// Mitsubishi GX Works2 project: 增加消防20180613   PLC: FX3G

PROGRAM MAIN
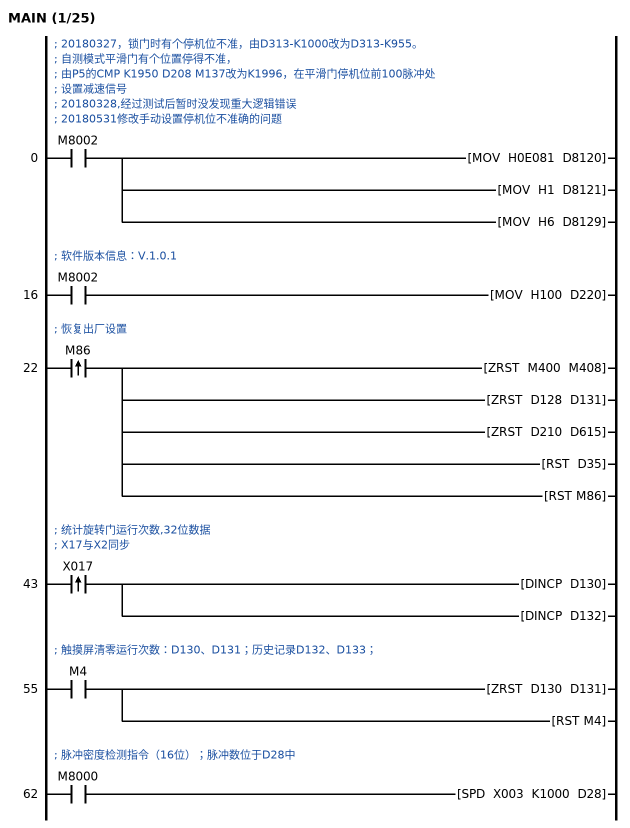
; 20180327，锁门时有个停机位不准，由D313-K1000改为D313-K955。
; 自测模式平滑门有个位置停得不准，
; 由P5的CMP K1950 D208 M137改为K1996，在平滑门停机位前100脉冲处
; 设置减速信号
; 20180328,经过测试后暂时没发现重大逻辑错误
; 20180531修改手动设置停机位不准确的问题
0     LD      M8002
      MOV     H0E081 D8120
        [note] 设置通讯方式
      MOV     H1 D8121
        [note] 站号设置：01H
      MOV     H6 D8129
        [note] 超时检查时间60ms
; 软件版本信息：V.1.0.1
16    LD      M8002
      MOV     H100 D220
        [note] V.1.0.1
; 恢复出厂设置
22    LDP     M86
      ZRST    M400 M408
      ZRST    D128 D131
      ZRST    D210 D615
      RST     D35
      RST     M86
; 统计旋转门运行次数,32位数据
; X17与X2同步
43    LDP     X017
      DINCP   D130
      DINCP   D132
; 触摸屏清零运行次数：D130、D131；历史记录D132、D133；
55    LD      M4
      ZRST    D130 D131
      RST     M4
; 脉冲密度检测指令（16位）；脉冲数位于D28中
62    LD      M8000
      SPD     X003 K1000 D28
        [note] 速度检测
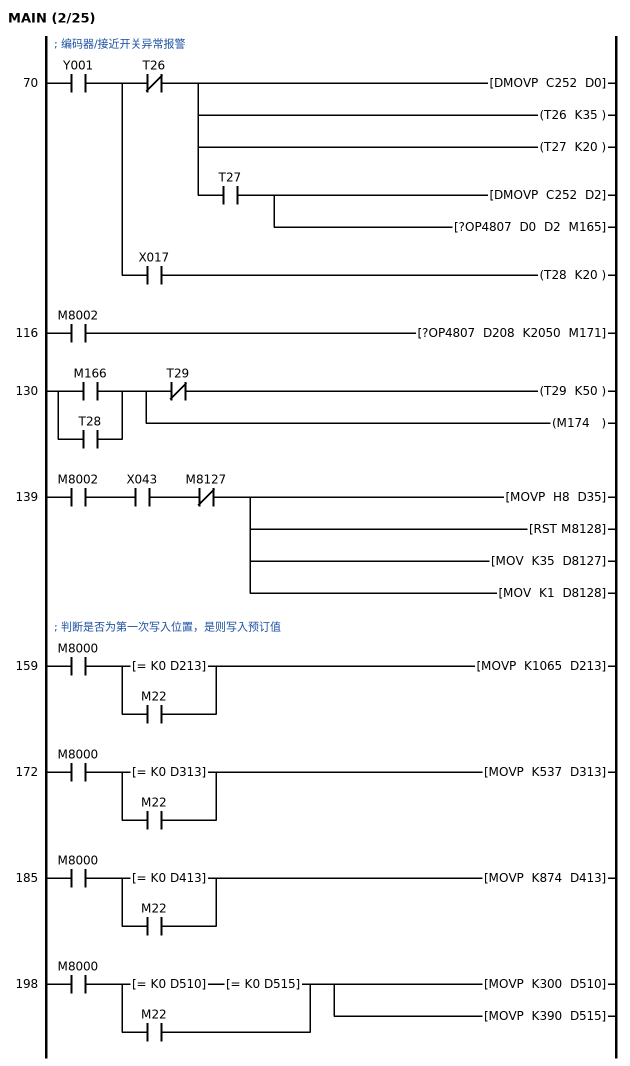
; 编码器/接近开关异常报警
70    LD      Y001
      MPS
      ANI     T26
      DMOVP   C252 D0
      OUT     T26 K35
      OUT     T27 K20
      AND     T27
      DMOVP   C252 D2
      ?OP4807 D0 D2 M165
        [note] Y1=1时，D0D1=D2D3，编码器坏
      MPP
      AND     X017
      OUT     T28 K20
        [note] Y1=1时，编码器连续2s清零0，坏
116   LD      M8002
      ?OP4807 D208 K2050 M171
        [note] 编码器值>2050时M173置位
130   LD      M166
      OR      T28
      MPS
      ANI     T29
      OUT     T29 K50
        [note] 每隔5秒发送一次报警命令
      MPP
      OUT     M174
139   LD      M8002
      AND     X043
      ANI     M8127
      MOVP    H8 D35
      RST     M8128
      MOV     K35 D8127
      MOV     K1 D8128
; 判断是否为第一次写入位置，是则写入预订值
159   LD      M8000
      LD=     K0 D213
      OR      M22
      ANB
      MOVP    K1065 D213
        [note] 平滑门位置
172   LD      M8000
      LD=     K0 D313
      OR      M22
      ANB
      MOVP    K537 D313
        [note] 冬季位置
185   LD      M8000
      LD=     K0 D413
      OR      M22
      ANB
      MOVP    K874 D413
        [note] 夏季位置
198   LD      M8000
      LD=     K0 D510
      AND=    K0 D515
      OR      M22
      ANB
      MOVP    K300 D510
        [note] 危险区域1
      MOVP    K390 D515
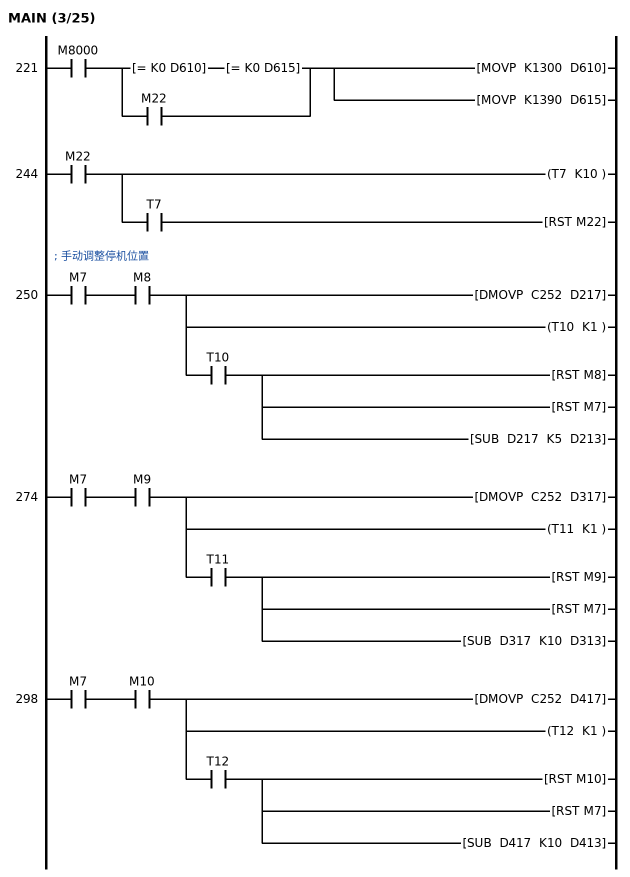
221   LD      M8000
      LD=     K0 D610
      AND=    K0 D615
      OR      M22
      ANB
      MOVP    K1300 D610
        [note] 危险区域2
      MOVP    K1390 D615
244   LD      M22
      OUT     T7 K10
      AND     T7
      RST     M22
; 手动调整停机位置
250   LD      M7
      AND     M8
      DMOVP   C252 D217
        [note] 手动调整平滑模式参考位
      OUT     T10 K1
      AND     T10
      RST     M8
      RST     M7
      SUB     D217 K5 D213
274   LD      M7
      AND     M9
      DMOVP   C252 D317
        [note] 手动调整冬季模式参考位
      OUT     T11 K1
      AND     T11
      RST     M9
      RST     M7
      SUB     D317 K10 D313
298   LD      M7
      AND     M10
      DMOVP   C252 D417
        [note] 手动调整夏季模式参考位
      OUT     T12 K1
      AND     T12
      RST     M10
      RST     M7
      SUB     D417 K10 D413
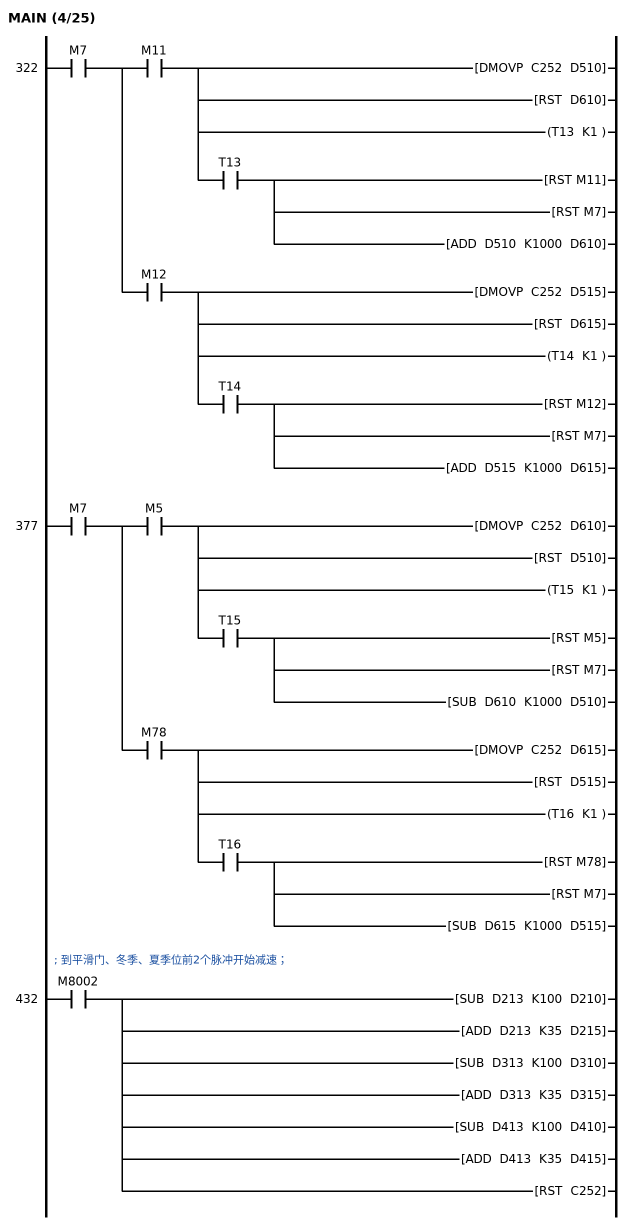
322   LD      M7
      MPS
      AND     M11
      DMOVP   C252 D510
        [note] 手动调危险区1参考位
      RST     D610
      OUT     T13 K1
      AND     T13
      RST     M11
      RST     M7
      ADD     D510 K1000 D610
      MPP
      AND     M12
      DMOVP   C252 D515
      RST     D615
      OUT     T14 K1
      AND     T14
      RST     M12
      RST     M7
      ADD     D515 K1000 D615
377   LD      M7
      MPS
      AND     M5
      DMOVP   C252 D610
        [note] 手动调危险区2参考位
      RST     D510
      OUT     T15 K1
      AND     T15
      RST     M5
      RST     M7
      SUB     D610 K1000 D510
      MPP
      AND     M78
      DMOVP   C252 D615
      RST     D515
      OUT     T16 K1
      AND     T16
      RST     M78
      RST     M7
      SUB     D615 K1000 D515
; 到平滑门、冬季、夏季位前2个脉冲开始减速；
432   LD      M8002
      SUB     D213 K100 D210
        [note] 确定参考位提前减速点
      ADD     D213 K35 D215
      SUB     D313 K100 D310
      ADD     D313 K35 D315
      SUB     D413 K100 D410
      ADD     D413 K35 D415
      RST     C252
        [note] 第一扫描周期编码器计数器清零
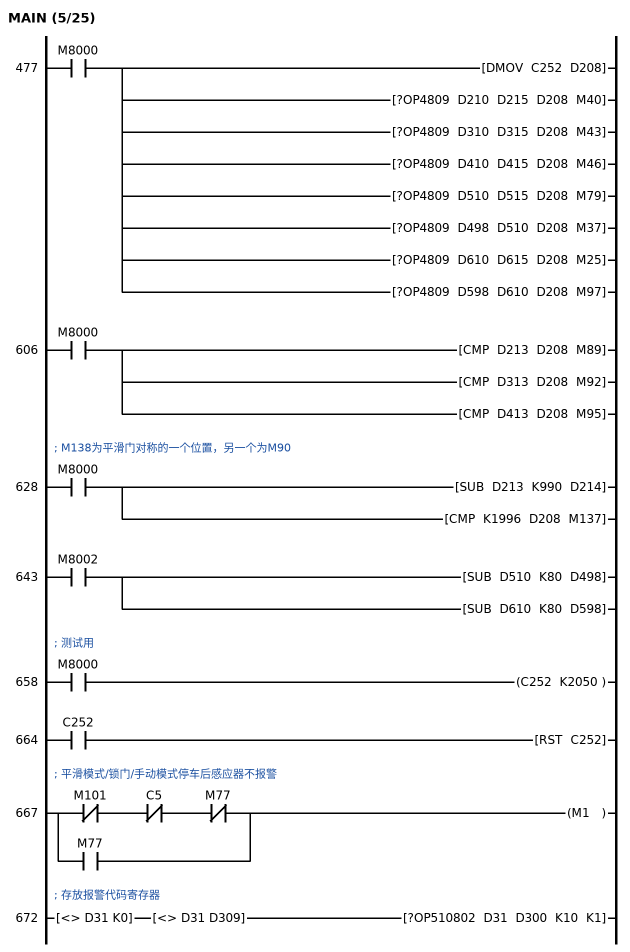
477   LD      M8000
      DMOV    C252 D208
      ?OP4809 D210 D215 D208 M40
        [note] 平滑门位置（199°）
      ?OP4809 D310 D315 D208 M43
        [note] M44：冬季位置（90°）
      ?OP4809 D410 D415 D208 M46
        [note] M47：夏季位置前减速标志（180°）
      ?OP4809 D510 D515 D208 M79
        [note] 危险区域1（76°-90°）
      ?OP4809 D498 D510 D208 M37
        [note] 危险区1减速带起点数据D498
      ?OP4809 D610 D615 D208 M25
        [note] 危险区域2（256°-270°）
      ?OP4809 D598 D610 D208 M97
        [note] 危险区2减速带起点数据D598
606   LD      M8000
      CMP     D213 D208 M89
        [note] 平滑门停机位
      CMP     D313 D208 M92
        [note] 冬季停机位
      CMP     D413 D208 M95
        [note] 夏季停机位
; M138为平滑门对称的一个位置，另一个为M90
628   LD      M8000
      SUB     D213 K990 D214
      CMP     K1996 D208 M137
643   LD      M8002
      SUB     D510 K80 D498
        [note] 危险区1-2个脉冲=减速带起点
      SUB     D610 K80 D598
        [note] 危险区2-2个脉冲=减速带起点
; 测试用
658   LD      M8000
      OUT     C252 K2050
664   LD      C252
      RST     C252
; 平滑模式/锁门/手动模式停车后感应器不报警
667   LDI     M101
      ANI     C5
      ANI     M77
      OR      M77
      OUT     M1
; 存放报警代码寄存器
672   LD<>    D31 K0
      AND<>   D31 D309
      ?OP510802 D31 D300 K10 K1
        [note] 有报警且不等于上次时移位
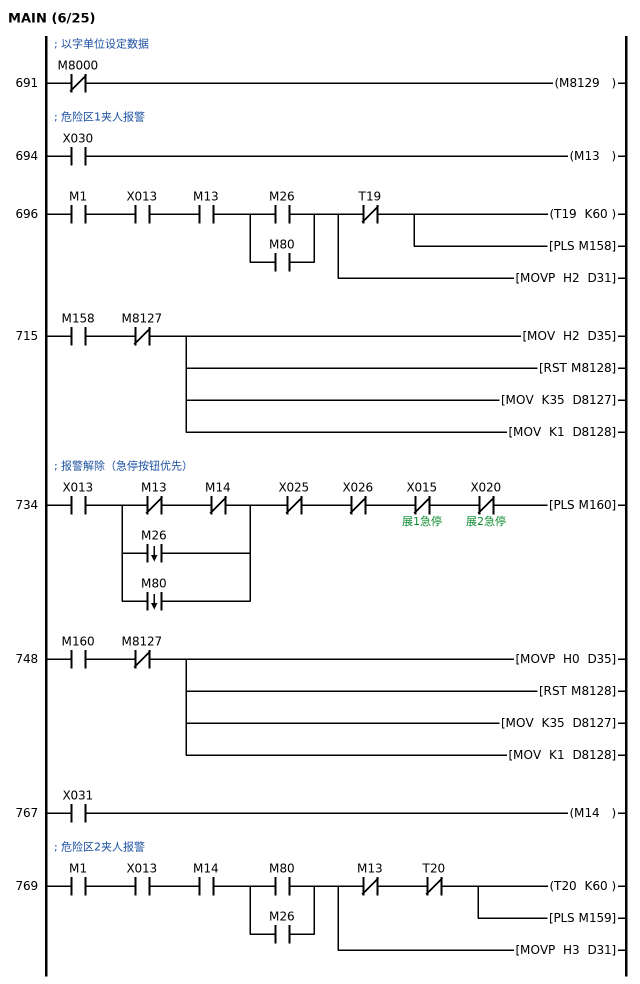
; 以字单位设定数据
691   LDI     M8000
      OUT     M8129
; 危险区1夹人报警
694   LD      X030
      OUT     M13
696   LD      M1
      AND     X013
      AND     M13
      LD      M26
      OR      M80
      ANB
      MPS
      ANI     T19
      OUT     T19 K60
        [note] 每隔1秒发送一次数据
      PLS     M158
      MPP
      MOVP    H2 D31
        [note] 报警代码
715   LD      M158
      ANI     M8127
      MOV     H2 D35
      RST     M8128
      MOV     K35 D8127
      MOV     K1 D8128
; 报警解除（急停按钮优先）
734   LD      X013
      LDI     M13
      ANI     M14
      ORF     M26
      ORF     M80
      ANB
      ANI     X025
      ANI     X026
      ANI     X015  ; 展1急停
      ANI     X020  ; 展2急停
      PLS     M160
748   LD      M160
      ANI     M8127
      MOVP    H0 D35
      RST     M8128
      MOV     K35 D8127
      MOV     K1 D8128
767   LD      X031
      OUT     M14
; 危险区2夹人报警
769   LD      M1
      AND     X013
      AND     M14
      LD      M80
      OR      M26
      ANB
      MPS
      ANI     M13
      ANI     T20
      OUT     T20 K60
        [note] 每隔6秒发送一次数据
      PLS     M159
      MPP
      MOVP    H3 D31
        [note] 报警代码
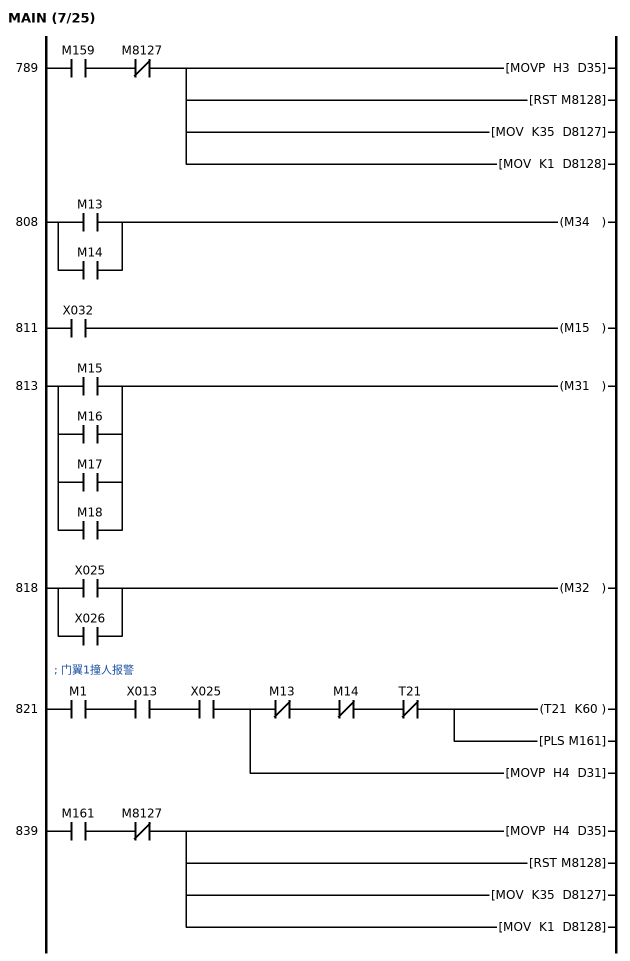
789   LD      M159
      ANI     M8127
      MOVP    H3 D35
      RST     M8128
      MOV     K35 D8127
      MOV     K1 D8128
808   LD      M13
      OR      M14
      OUT     M34
        [note] 危险区传感器启动信号
811   LD      X032
      OUT     M15
813   LD      M15
      OR      M16
      OR      M17
      OR      M18
      OUT     M31
        [note] 启动传感器信号
818   LD      X025
      OR      X026
      OUT     M32
        [note] 门翼急停信号
; 门翼1撞人报警
821   LD      M1
      AND     X013
      AND     X025
      MPS
      ANI     M13
      ANI     M14
      ANI     T21
      OUT     T21 K60
        [note] 每隔6秒发送一次数据
      PLS     M161
      MPP
      MOVP    H4 D31
        [note] 报警代码
839   LD      M161
      ANI     M8127
      MOVP    H4 D35
      RST     M8128
      MOV     K35 D8127
      MOV     K1 D8128
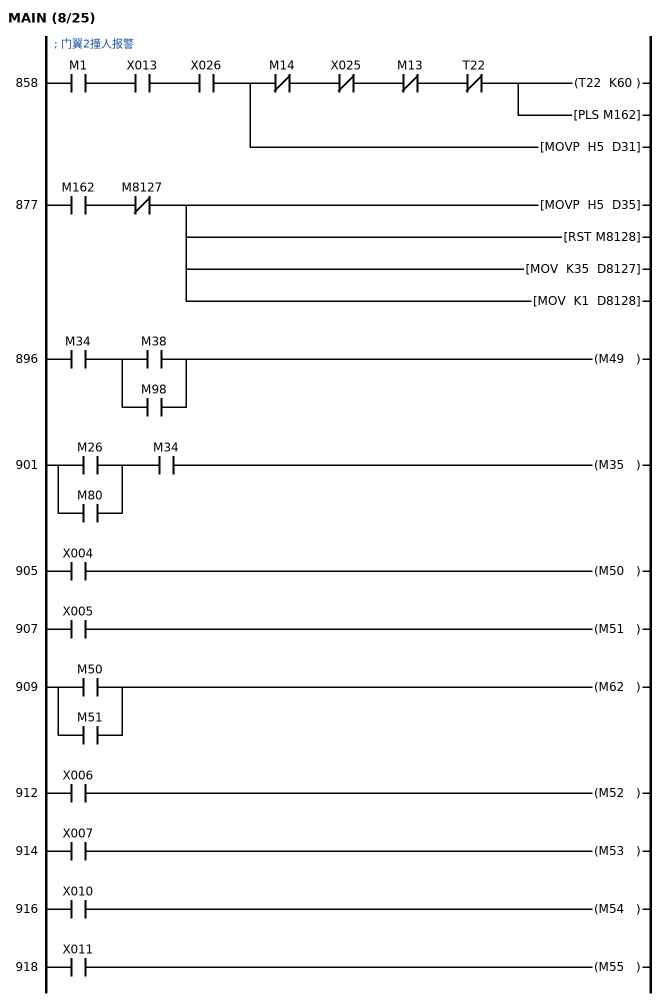
; 门翼2撞人报警
858   LD      M1
      AND     X013
      AND     X026
      MPS
      ANI     M14
      ANI     X025
      ANI     M13
      ANI     T22
      OUT     T22 K60
        [note] 每隔6秒发送一次数据
      PLS     M162
      MPP
      MOVP    H5 D31
877   LD      M162
      ANI     M8127
      MOVP    H5 D35
      RST     M8128
      MOV     K35 D8127
      MOV     K1 D8128
896   LD      M34
      LD      M38
      OR      M98
      ANB
      OUT     M49
        [note] 危险区前减速带有信号标示
901   LD      M26
      OR      M80
      AND     M34
      OUT     M35
        [note] 危险区信号标示
905   LD      X004
      OUT     M50
        [note] 平滑门室内启动传感器
907   LD      X005
      OUT     M51
        [note] 平滑门室外启动传感器
909   LD      M50
      OR      M51
      OUT     M62
        [note] 平滑门启动传感器
912   LD      X006
      OUT     M52
        [note] 门翼1慢速
914   LD      X007
      OUT     M53
        [note] 门翼1急停
916   LD      X010
      OUT     M54
        [note] 门翼2慢速
918   LD      X011
      OUT     M55
        [note] 门翼2急停
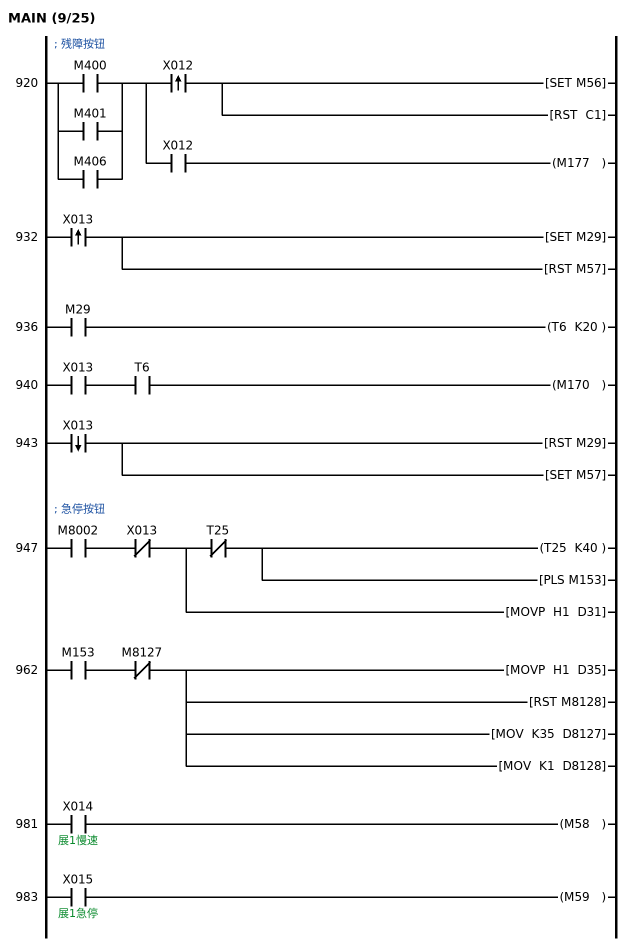
; 残障按钮
920   LD      M400
      OR      M401
      OR      M406
      MPS
      ANDP    X012
      SET     M56
      RST     C1
      MPP
      AND     X012
      OUT     M177
        [note] 残障按钮一直按下，慢速
932   LDP     X013
      SET     M29
      RST     M57
936   LD      M29
      OUT     T6 K20
940   LD      X013
      AND     T6
      OUT     M170
943   LDF     X013
      RST     M29
      SET     M57
; 急停按钮
947   LD      M8002
      ANI     X013
      MPS
      ANI     T25
      OUT     T25 K40
      PLS     M153
      MPP
      MOVP    H1 D31
        [note] 报警代码
962   LD      M153
      ANI     M8127
      MOVP    H1 D35
      RST     M8128
      MOV     K35 D8127
      MOV     K1 D8128
981   LD      X014  ; 展1慢速
      OUT     M58
983   LD      X015  ; 展1急停
      OUT     M59
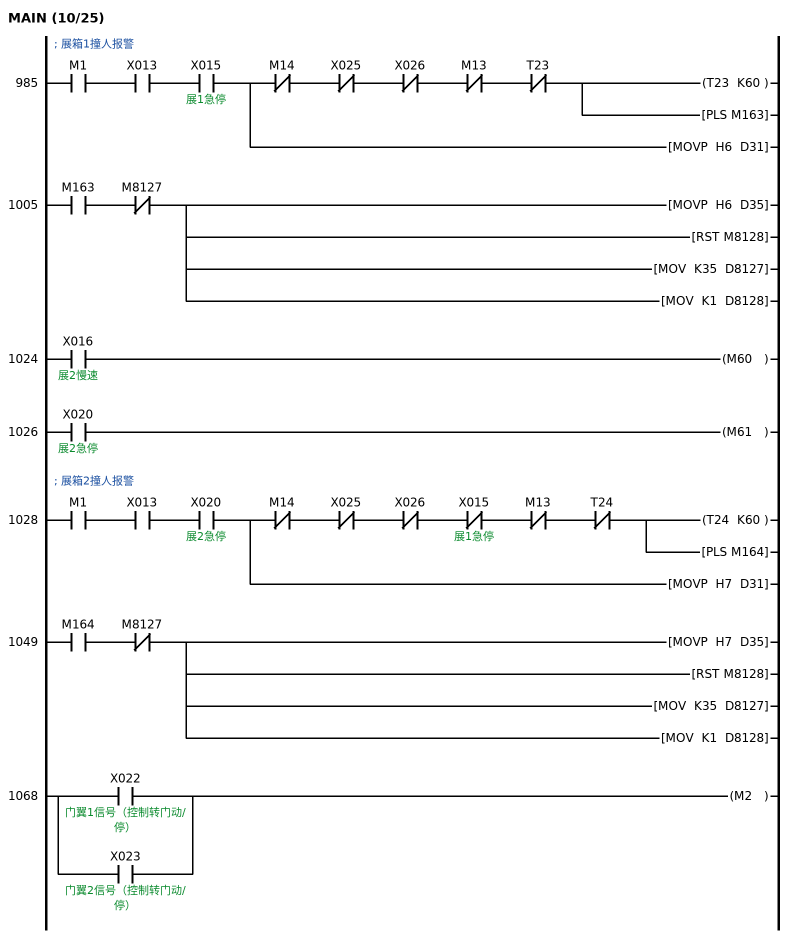
; 展箱1撞人报警
985   LD      M1
      AND     X013
      AND     X015  ; 展1急停
      MPS
      ANI     M14
      ANI     X025
      ANI     X026
      ANI     M13
      ANI     T23
      OUT     T23 K60
      PLS     M163
      MPP
      MOVP    H6 D31
        [note] 报警代码
1005  LD      M163
      ANI     M8127
      MOVP    H6 D35
      RST     M8128
      MOV     K35 D8127
      MOV     K1 D8128
1024  LD      X016  ; 展2慢速
      OUT     M60
1026  LD      X020  ; 展2急停
      OUT     M61
; 展箱2撞人报警
1028  LD      M1
      AND     X013
      AND     X020  ; 展2急停
      MPS
      ANI     M14
      ANI     X025
      ANI     X026
      ANI     X015  ; 展1急停
      ANI     M13
      ANI     T24
      OUT     T24 K60
      PLS     M164
      MPP
      MOVP    H7 D31
1049  LD      M164
      ANI     M8127
      MOVP    H7 D35
      RST     M8128
      MOV     K35 D8127
      MOV     K1 D8128
1068  LD      X022  ; 门翼1信号（控制转门动/停）
      OR      X023  ; 门翼2信号（控制转门动/停）
      OUT     M2
        [note] 门翼控制器信号--控制Y1
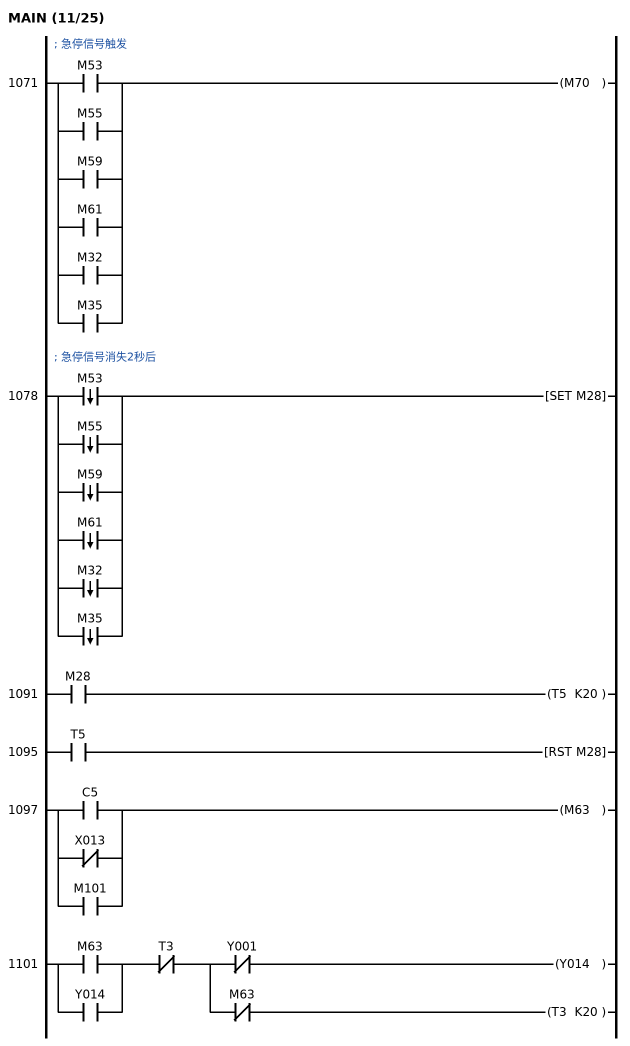
; 急停信号触发
1071  LD      M53
      OR      M55
      OR      M59
      OR      M61
      OR      M32
      OR      M35
      OUT     M70
; 急停信号消失2秒后
1078  LDF     M53
      ORF     M55
      ORF     M59
      ORF     M61
      ORF     M32
      ORF     M35
      SET     M28
1091  LD      M28
      OUT     T5 K20
1095  LD      T5
      RST     M28
1097  LD      C5
      ORI     X013
      OR      M101
      OUT     M63
        [note] 锁门/急停/平滑到位启动刹车
1101  LD      M63
      OR      Y014
      ANI     T3
      MPS
      ANI     Y001
      OUT     Y014
        [note] 刹车信号
      MPP
      ANI     M63
      OUT     T3 K20
        [note] 信号消失后延时2秒
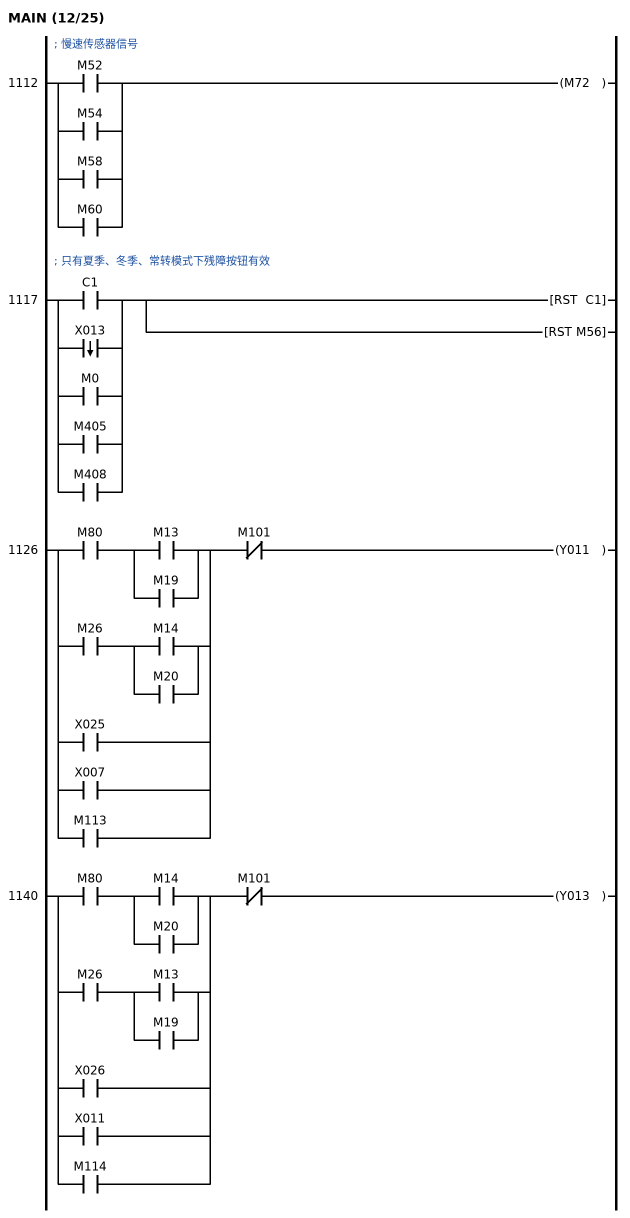
; 慢速传感器信号
1112  LD      M52
      OR      M54
      OR      M58
      OR      M60
      OUT     M72
; 只有夏季、冬季、常转模式下残障按钮有效
1117  LD      C1
      ORF     X013
      OR      M0
      OR      M405
      OR      M408
      RST     C1
      RST     M56
1126  LD      M80
      LD      M13
      OR      M19
      ANB
      LD      M26
      LD      M14
      OR      M20
      ANB
      ORB
      OR      X025
      OR      X007
      OR      M113
      ANI     M101
      OUT     Y011
        [note] 门翼1后退信号
1140  LD      M80
      LD      M14
      OR      M20
      ANB
      LD      M26
      LD      M13
      OR      M19
      ANB
      ORB
      OR      X026
      OR      X011
      OR      M114
      ANI     M101
      OUT     Y013
        [note] 门翼2后退信号
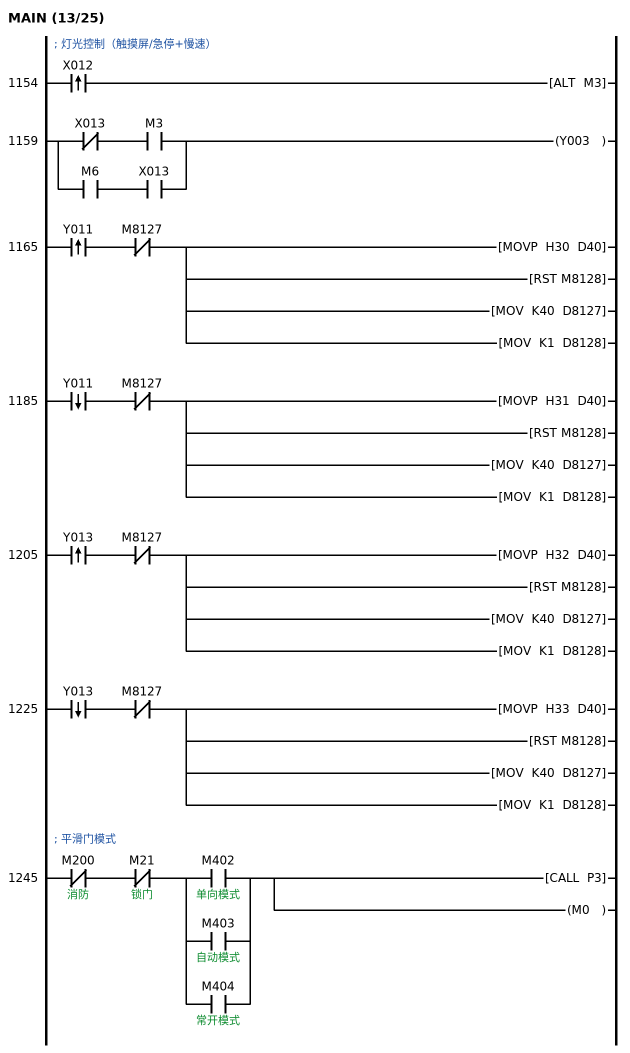
; 灯光控制（触摸屏/急停+慢速）
1154  LDP     X012
      ALT     M3
1159  LDI     X013
      AND     M3
      LD      M6
      AND     X013
      ORB
      OUT     Y003
        [note] LED灯光
1165  LDP     Y011
      ANI     M8127
      MOVP    H30 D40
        [note] 门翼1后退信息
      RST     M8128
      MOV     K40 D8127
      MOV     K1 D8128
1185  LDF     Y011
      ANI     M8127
      MOVP    H31 D40
        [note] 门翼1关闭信息
      RST     M8128
      MOV     K40 D8127
      MOV     K1 D8128
1205  LDP     Y013
      ANI     M8127
      MOVP    H32 D40
        [note] 门翼2后退信息
      RST     M8128
      MOV     K40 D8127
      MOV     K1 D8128
1225  LDF     Y013
      ANI     M8127
      MOVP    H33 D40
        [note] 门翼2后退信息
      RST     M8128
      MOV     K40 D8127
      MOV     K1 D8128
; 平滑门模式
1245  LDI     M200  ; 消防
      ANI     M21  ; 锁门
      LD      M402  ; 单向模式
      OR      M403  ; 自动模式
      OR      M404  ; 常开模式
      ANB
      CALL    P3
      OUT     M0
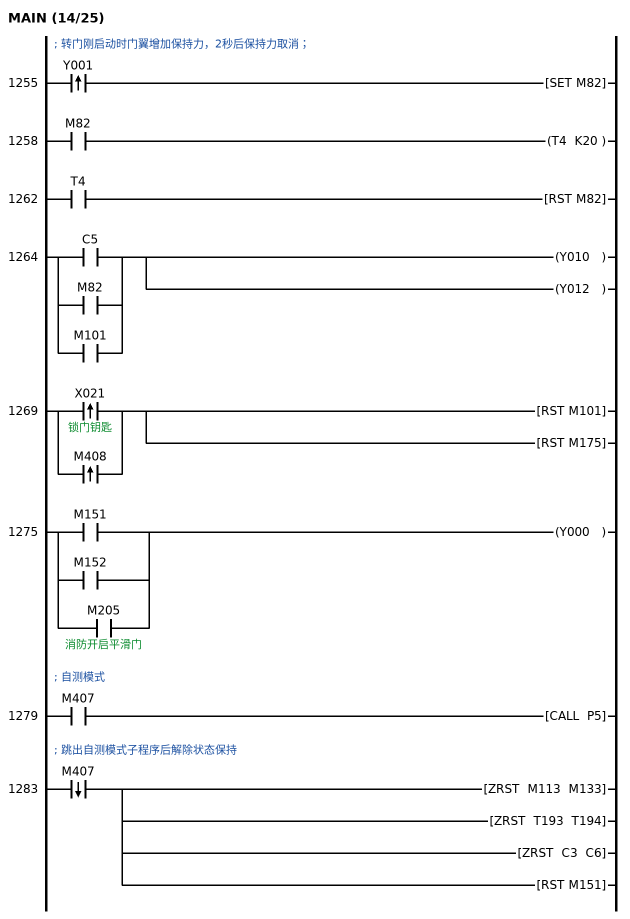
; 转门刚启动时门翼增加保持力，2秒后保持力取消；
1255  LDP     Y001
      SET     M82
1258  LD      M82
      OUT     T4 K20
1262  LD      T4
      RST     M82
1264  LD      C5
      OR      M82
      OR      M101
      OUT     Y010
        [note] 门翼1带保持力
      OUT     Y012
        [note] 门翼2带保持力
1269  LDP     X021  ; 锁门钥匙
      ORP     M408
      RST     M101
        [note] 锁门时，清除平滑模式标志位
      RST     M175
1275  LD      M151
      OR      M152
      OR      M205  ; 消防开启平滑门
      OUT     Y000
        [note] 平滑门开启
; 自测模式
1279  LD      M407
      CALL    P5
; 跳出自测模式子程序后解除状态保持
1283  LDF     M407
      ZRST    M113 M133
      ZRST    T193 T194
      ZRST    C3 C6
      RST     M151
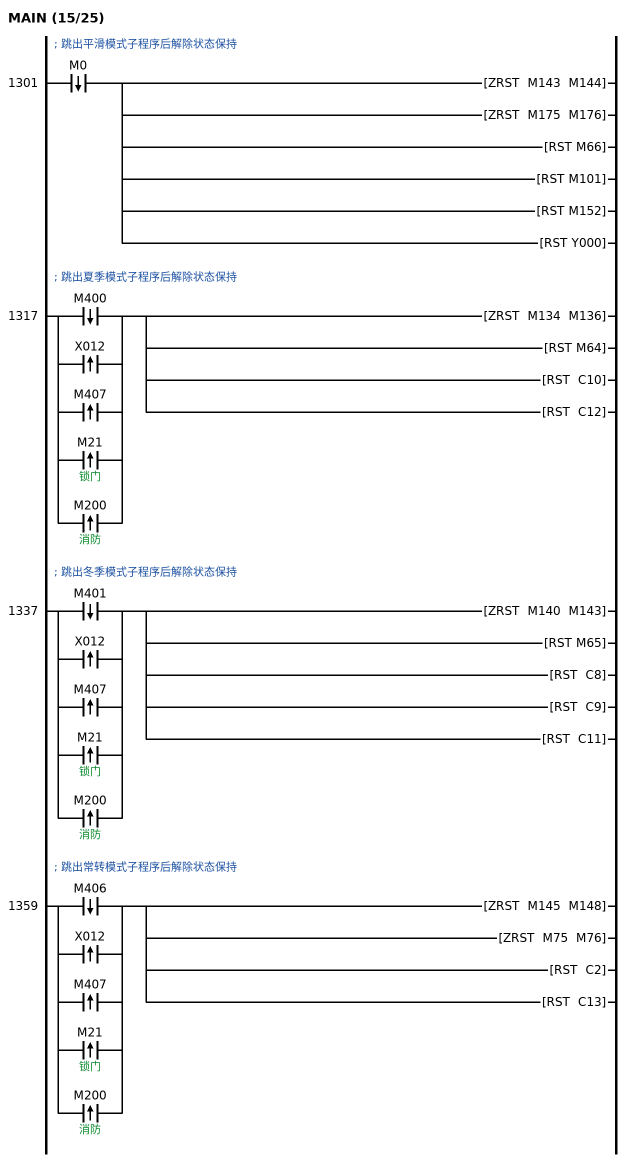
; 跳出平滑模式子程序后解除状态保持
1301  LDF     M0
      ZRST    M143 M144
      ZRST    M175 M176
      RST     M66
      RST     M101
      RST     M152
      RST     Y000
; 跳出夏季模式子程序后解除状态保持
1317  LDF     M400
      ORP     X012
      ORP     M407
      ORP     M21  ; 锁门
      ORP     M200  ; 消防
      ZRST    M134 M136
      RST     M64
      RST     C10
      RST     C12
; 跳出冬季模式子程序后解除状态保持
1337  LDF     M401
      ORP     X012
      ORP     M407
      ORP     M21  ; 锁门
      ORP     M200  ; 消防
      ZRST    M140 M143
      RST     M65
      RST     C8
      RST     C9
      RST     C11
; 跳出常转模式子程序后解除状态保持
1359  LDF     M406
      ORP     X012
      ORP     M407
      ORP     M21  ; 锁门
      ORP     M200  ; 消防
      ZRST    M145 M148
      ZRST    M75 M76
      RST     C2
      RST     C13
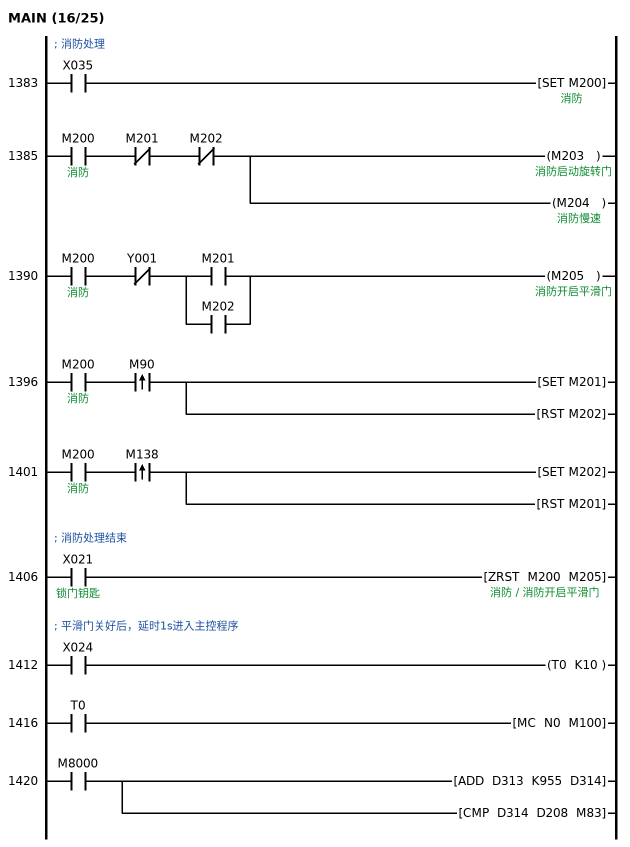
; 消防处理
1383  LD      X035
      SET     M200  ; 消防
        [note] 消防信号标志位置1
1385  LD      M200  ; 消防
      ANI     M201
      ANI     M202
      OUT     M203  ; 消防启动旋转门
        [note] 消防信号门启动：Y1
      OUT     M204  ; 消防慢速
        [note] 旋转门慢速：Y7
1390  LD      M200  ; 消防
      ANI     Y001
      LD      M201
      OR      M202
      ANB
      OUT     M205  ; 消防开启平滑门
        [note] 平滑门常开：Y0
1396  LD      M200  ; 消防
      ANDP    M90
      SET     M201
      RST     M202
1401  LD      M200  ; 消防
      ANDP    M138
      SET     M202
      RST     M201
; 消防处理结束
1406  LD      X021  ; 锁门钥匙
      ZRST    M200 M205
        [note] 锁门钥匙清除消防信号
; 平滑门关好后，延时1s进入主控程序
1412  LD      X024
      OUT     T0 K10
1416  LD      T0
      MC      N0 M100
        [note] 主控程序开始
1420  LD      M8000
      ADD     D313 K955 D314
        [note] 锁门位置，对称两位置都有效
      CMP     D314 D208 M83
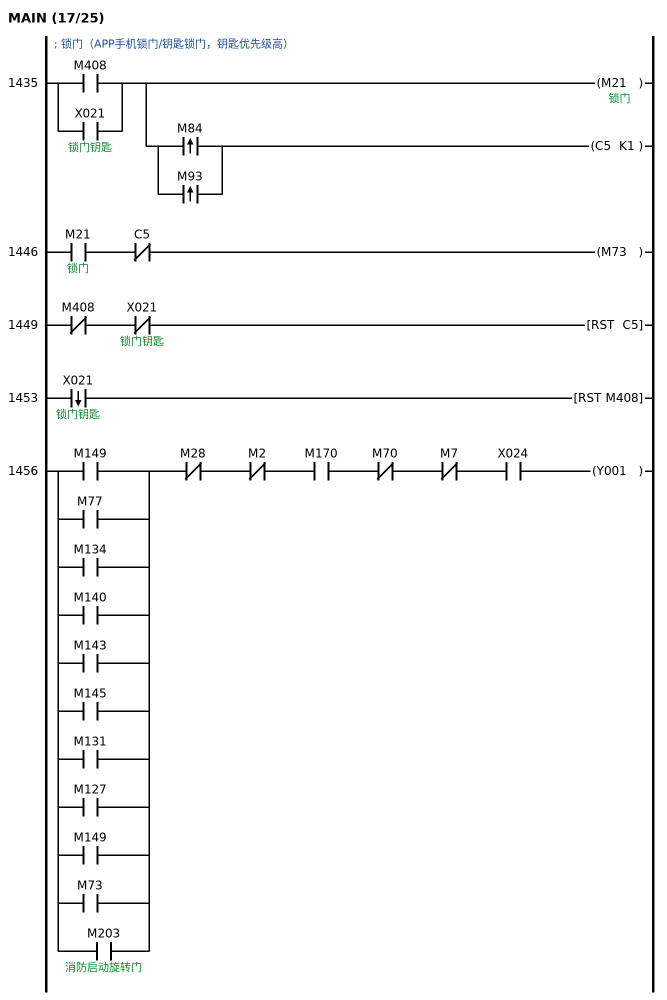
; 锁门（APP手机锁门/钥匙锁门，钥匙优先级高）
1435  LD      M408
      OR      X021  ; 锁门钥匙
      OUT     M21  ; 锁门
      LDP     M84
      ORP     M93
      ANB
      OUT     C5 K1
1446  LD      M21  ; 锁门
      ANI     C5
      OUT     M73
1449  LDI     M408
      ANI     X021  ; 锁门钥匙
      RST     C5
1453  LDF     X021  ; 锁门钥匙
      RST     M408
1456  LD      M149
      OR      M77
      OR      M134
      OR      M140
      OR      M143
      OR      M145
      OR      M131
      OR      M127
      OR      M149
      OR      M73
      OR      M203  ; 消防启动旋转门
      ANI     M28
      ANI     M2
      AND     M170
      ANI     M70
      ANI     M7
      AND     X024
      OUT     Y001
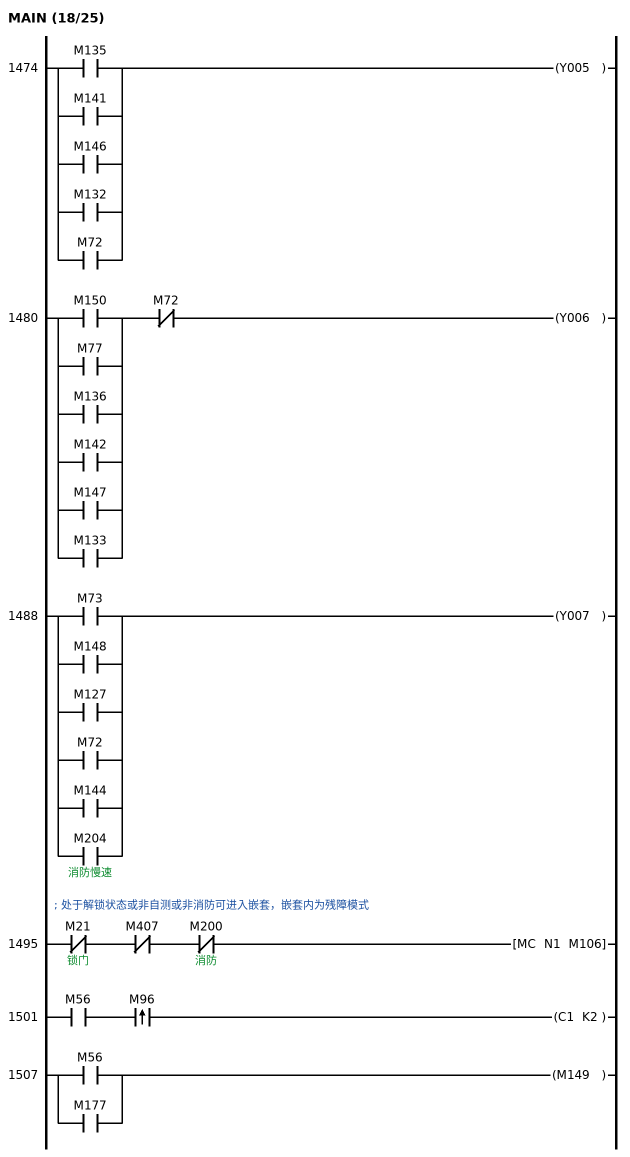
1474  LD      M135
      OR      M141
      OR      M146
      OR      M132
      OR      M72
      OUT     Y005
1480  LD      M150
      OR      M77
      OR      M136
      OR      M142
      OR      M147
      OR      M133
      ANI     M72
      OUT     Y006
1488  LD      M73
      OR      M148
      OR      M127
      OR      M72
      OR      M144
      OR      M204  ; 消防慢速
      OUT     Y007
; 处于解锁状态或非自测或非消防可进入嵌套，嵌套内为残障模式
1495  LDI     M21  ; 锁门
      ANI     M407
      ANI     M200  ; 消防
      MC      N1 M106
1501  LD      M56
      ANDP    M96
      OUT     C1 K2
1507  LD      M56
      OR      M177
      OUT     M149
        [note] 启动：Y1
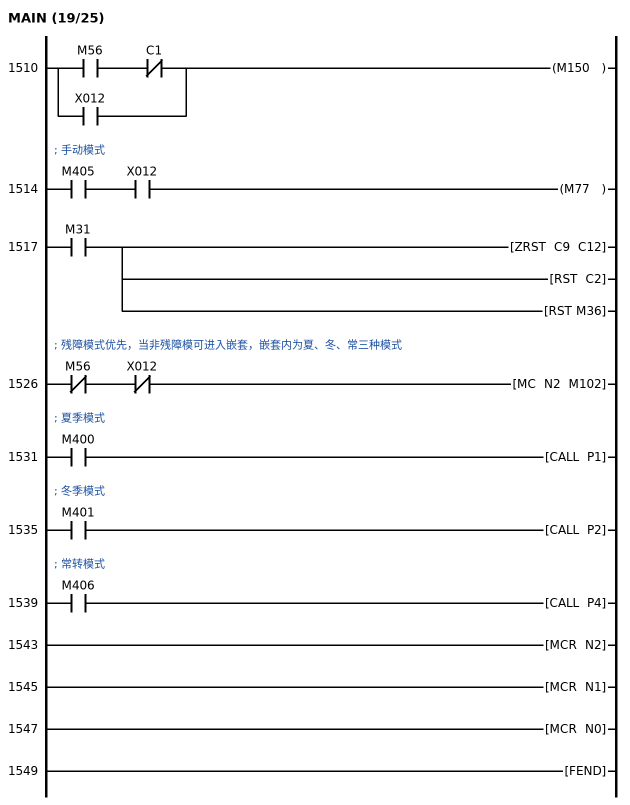
1510  LD      M56
      ANI     C1
      OR      X012
      OUT     M150
        [note] 低速：Y6
; 手动模式
1514  LD      M405
      AND     X012
      OUT     M77
1517  LD      M31
      ZRST    C9 C12
      RST     C2
      RST     M36
; 残障模式优先，当非残障模可进入嵌套，嵌套内为夏、冬、常三种模式
1526  LDI     M56
      ANI     X012
      MC      N2 M102
; 夏季模式
1531  LD      M400
      CALL    P1
; 冬季模式
1535  LD      M401
      CALL    P2
; 常转模式
1539  LD      M406
      CALL    P4
1543  MCR     N2
1545  MCR     N1
1547  MCR     N0
        [note] 主控程序结束
1549  FEND
        [note] 主程序结束
      P1
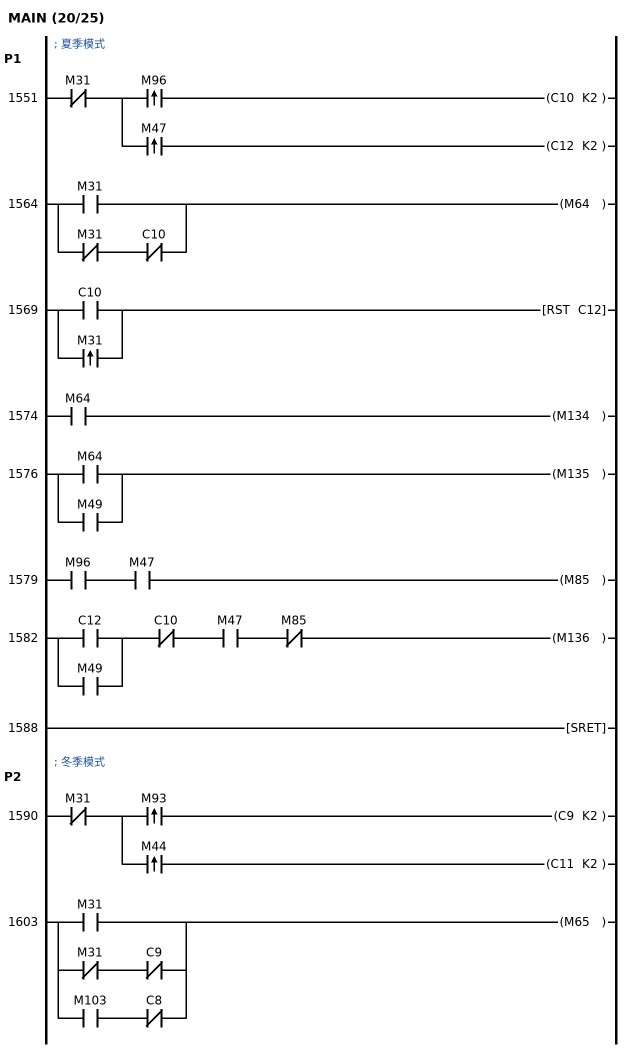
; 夏季模式
1551  LDI     M31
      MPS
      ANDP    M96
      OUT     C10 K2
      MPP
      ANDP    M47
      OUT     C12 K2
1564  LD      M31
      LDI     M31
      ANI     C10
      ORB
      OUT     M64
1569  LD      C10
      ORP     M31
      RST     C12
1574  LD      M64
      OUT     M134
        [note] 启动：Y1
1576  LD      M64
      OR      M49
      OUT     M135
        [note] 中速：Y5
1579  LD      M96
      AND     M47
      OUT     M85
1582  LD      C12
      OR      M49
      ANI     C10
      AND     M47
      ANI     M85
      OUT     M136
        [note] 低速：Y6
1588  SRET
      P2
; 冬季模式
1590  LDI     M31
      MPS
      ANDP    M93
      OUT     C9 K2
      MPP
      ANDP    M44
      OUT     C11 K2
1603  LD      M31
      LDI     M31
      ANI     C9
      ORB
      LD      M103
      ANI     C8
      ORB
      OUT     M65
        [note] 启动信号/消失后转2圈/防冬季被困
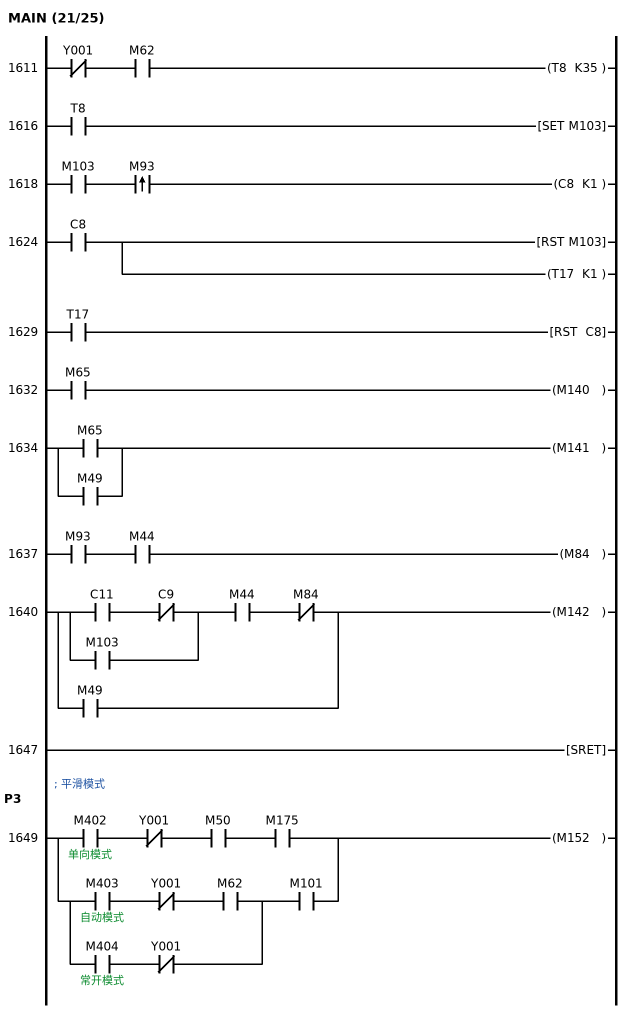
1611  LDI     Y001
      AND     M62
      OUT     T8 K35
1616  LD      T8
      SET     M103
1618  LD      M103
      ANDP    M93
      OUT     C8 K1
1624  LD      C8
      RST     M103
      OUT     T17 K1
1629  LD      T17
      RST     C8
1632  LD      M65
      OUT     M140
        [note] 启动：Y1
1634  LD      M65
      OR      M49
      OUT     M141
        [note] 高速：Y5
1637  LD      M93
      AND     M44
      OUT     M84
1640  LD      C11
      ANI     C9
      OR      M103
      AND     M44
      ANI     M84
      OR      M49
      OUT     M142
        [note] 低速：Y6
1647  SRET
      P3
; 平滑模式
1649  LD      M402  ; 单向模式
      ANI     Y001
      AND     M50
      AND     M175
      LD      M403  ; 自动模式
      ANI     Y001
      AND     M62
      LD      M404  ; 常开模式
      ANI     Y001
      ORB
      AND     M101
      ORB
      OUT     M152
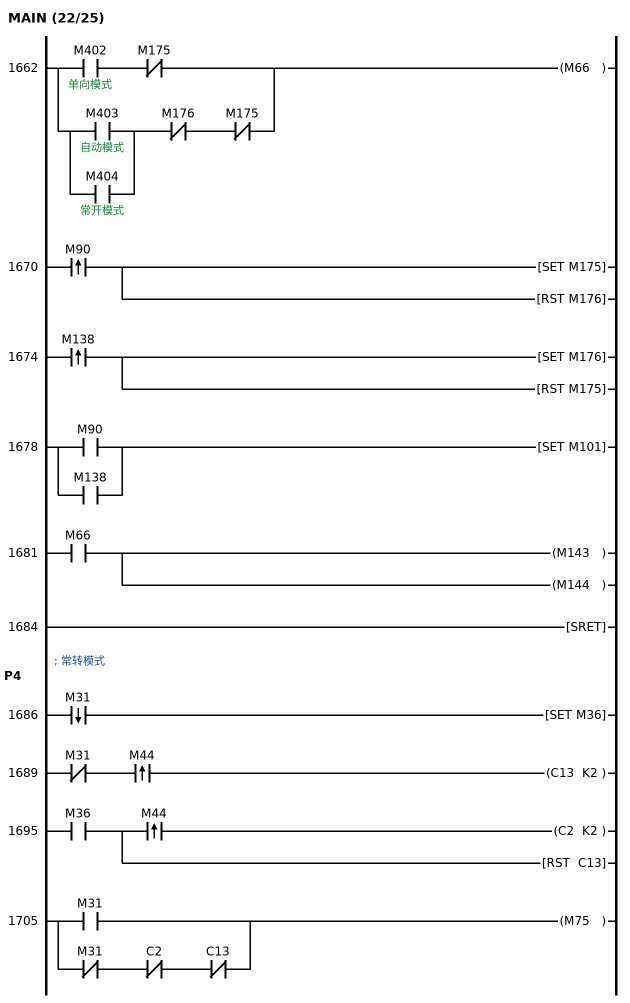
1662  LD      M402  ; 单向模式
      ANI     M175
      LD      M403  ; 自动模式
      OR      M404  ; 常开模式
      ANI     M176
      ANI     M175
      ORB
      OUT     M66
1670  LDP     M90
      SET     M175
      RST     M176
1674  LDP     M138
      SET     M176
      RST     M175
1678  LD      M90
      OR      M138
      SET     M101
1681  LD      M66
      OUT     M143
        [note] 启动：Y1
      OUT     M144
        [note] 慢速：Y7
1684  SRET
      P4
; 常转模式
1686  LDF     M31
      SET     M36
1689  LDI     M31
      ANDP    M44
      OUT     C13 K2
1695  LD      M36
      MPS
      ANDP    M44
      OUT     C2 K2
      MPP
      RST     C13
1705  LD      M31
      LDI     M31
      ANI     C2
      ANI     C13
      ORB
      OUT     M75
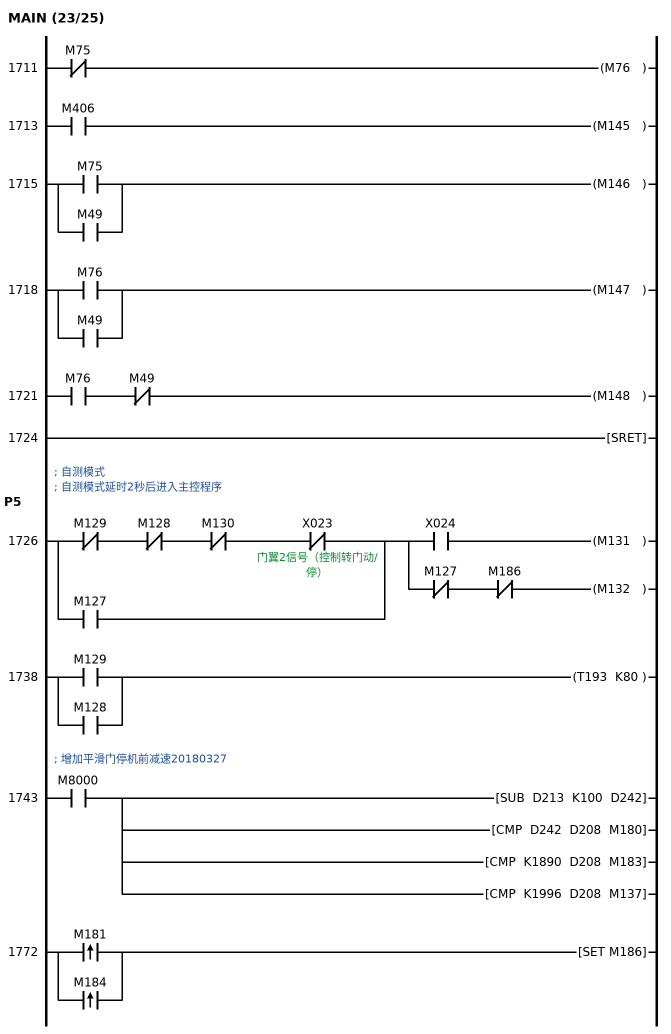
1711  LDI     M75
      OUT     M76
1713  LD      M406
      OUT     M145
        [note] 启动：Y1
1715  LD      M75
      OR      M49
      OUT     M146
        [note] 高速：Y5
1718  LD      M76
      OR      M49
      OUT     M147
        [note] 低速：Y6
1721  LD      M76
      ANI     M49
      OUT     M148
        [note] 低速：Y7
1724  SRET
      P5
; 自测模式
; 自测模式延时2秒后进入主控程序
1726  LDI     M129
      ANI     M128
      ANI     M130
      ANI     X023  ; 门翼2信号（控制转门动/停）
      OR      M127
      MPS
      AND     X024
      OUT     M131
        [note] 旋转门启动：Y1
      MPP
      ANI     M127
      ANI     M186
      OUT     M132
        [note] 高速运行：Y5
1738  LD      M129
      OR      M128
      OUT     T193 K80
        [note] 到夏/冬季停机位时停止8秒
; 增加平滑门停机前减速20180327
1743  LD      M8000
      SUB     D213 K100 D242
      CMP     D242 D208 M180
        [note] 自测模式平滑门位置前100减速
      CMP     K1890 D208 M183
        [note] 平滑门位置对称一侧前100减速
      CMP     K1996 D208 M137
1772  LDP     M181
      ORP     M184
      SET     M186
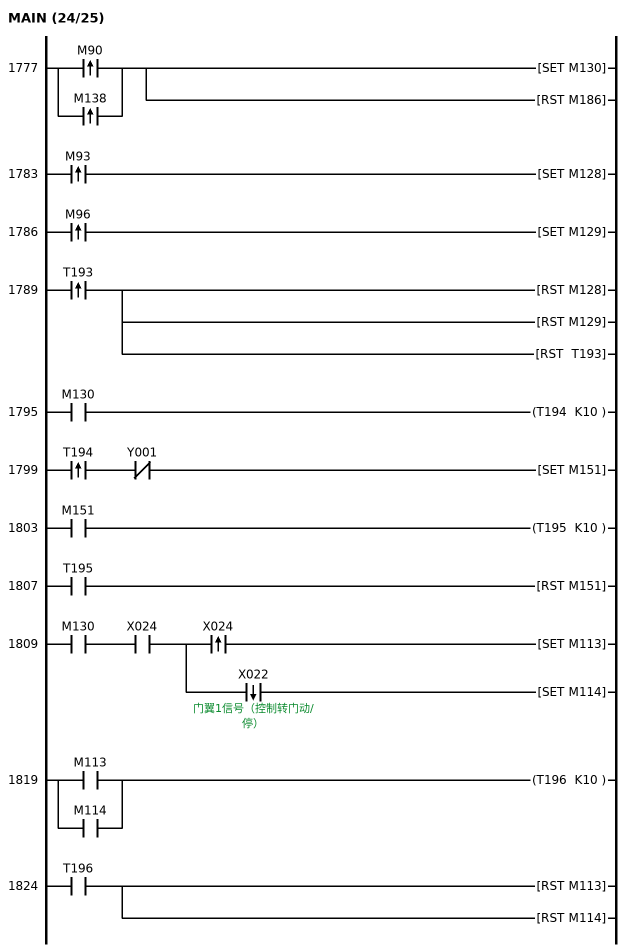
1777  LDP     M90
      ORP     M138
      SET     M130
        [note] 平滑门停机位时：M130=1
      RST     M186
1783  LDP     M93
      SET     M128
        [note] 冬季停机位时：M128=1
1786  LDP     M96
      SET     M129
        [note] 夏季停机位时：M129=1
1789  LDP     T193
      RST     M128
      RST     M129
      RST     T193
1795  LD      M130
      OUT     T194 K10
1799  LDP     T194
      ANI     Y001
      SET     M151
        [note] 到平滑门位置后延时1秒开门：Y0=1
1803  LD      M151
      OUT     T195 K10
1807  LD      T195
      RST     M151
1809  LD      M130
      AND     X024
      MPS
      ANDP    X024
      SET     M113
        [note] 门翼1开启
      MPP
      ANDF    X022  ; 门翼1信号（控制转门动/停）
      SET     M114
        [note] 门翼2开启
1819  LD      M113
      OR      M114
      OUT     T196 K10
1824  LD      T196
      RST     M113
      RST     M114
